// TIA Portal V20 export
// export: Created 2025-12-01T14:56:18.1563834Z, ExportSetting None, DisplayName Totally Integrated Automation Portal, DisplayVersion V20 Update 3, DisplayName TIA Portal Openness, DisplayVersion V20 Update 3, DisplayName TIA Portal Version Control Interface, DisplayVersion V20 Update 3, DisplayName STEP 7 Professional, DisplayVersion V20 Update 3, DisplayName STEP 7 Safety, DisplayVersion V20 Update 2, DisplayName WinCC Basic/Comfort/Advanced, DisplayVersion V20 Update 3, DisplayName WinCC Professional, DisplayVersion V20 Update 3, DisplayName WinCC Unified, DisplayVersion V20 Update 3
TYPE "Danfoss_Dig_Input_PN"
   STRUCT
      Reserved_1_0 : Bool;
      Reserved_1_1 : Bool;
      Reserved_1_2 : Bool;
      Reserved_1_3 : Bool;
      Reserved_1_4 : Bool;
      Reserved_1_5 : Bool;
      Reserved_1_6 : Bool;
      Reserved_1_7 : Bool;
      Dig_Input_33 : Bool;
      Dig_Input_32 : Bool;
      Dig_Input_29 : Bool;
      Dig_Input_27 : Bool;
      Dig_Input_19 : Bool;
      Dig_Input_18 : Bool;
      Reserved_6 : Bool;
      Reserved_7 : Bool;
   END_STRUCT;
END_TYPE
